FUNCTION AQ_5V : INT
VAR_INPUT
	Norm_input : REAL;
	x_max : REAL := 10;
	x_min : REAL := 0;
END_VAR
VAR
	voltage_reading : REAL;
END_VAR

voltage_reading := 5 * Norm_input;
AQ_5V := REAL_TO_INT (32767 * (voltage_reading - x_min) / (x_max - x_min));

END_FUNCTION

(* stored: Version 1.1.0.1, ProductVersion 3.1.4024.11
   POU AQ_5V: Id {7196eeea-21cb-421c-a821-2cdbae8393aa}, SpecialFunc None *)
